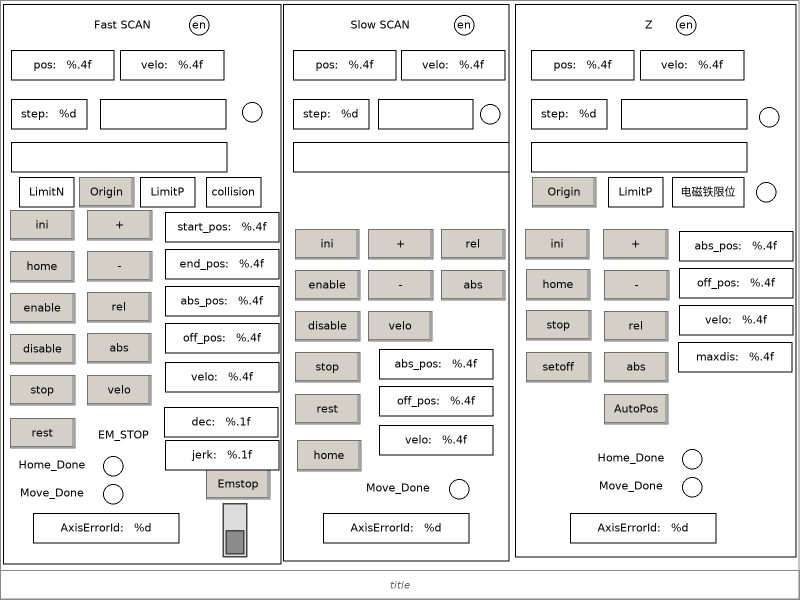
VISUALIZATION F1_AXIS  // 800x600
    RoundedRectangle (3,4 278x560)
    RoundedRectangle (515,4 281x553)
    RoundedRectangle (283,4 226x557)
    Button (87,210 65x30), "+", colour toggle: GVL_API.stAxis[1].JogForward
        tap GVL_API.stAxis[1].JogForward
    Button (87,251 65x30), "-", colour toggle: GVL_API.stAxis[1].JogBackwards
        tap GVL_API.stAxis[1].JogBackwards
    Button (10,251 64x31), "home", colour toggle: GVL_API.stAxis[1].homeExe
        toggle GVL_API.stAxis[1].homeExe
    Button (79,177 55x30), "Origin", colour toggle: Axis[1].IO.snHome
        toggle Axis[1].IO.snHome
    Rectangle (11,50 103x30), "pos: %.4f", text variable: Axis[1].Ref.NcToPlc.ActPos
    Rectangle (120,50 104x30), "velo: %.4f", text variable: Axis[1].Ref.NcToPlc.ActVelo
    Ellipse (189,15 20x20), "en", colour toggle: Axis[1].Ref.Status.ControlLoopClosed
    Button (87,292 64x30), "rel", colour toggle: GVL_API.stAxis[1].MoveRelativeExe
        toggle GVL_API.stAxis[1].MoveRelativeExe
    Button (87,333 64x30), "abs", colour toggle: GVL_API.stAxis[1].MoveAbsoluteExe
        toggle GVL_API.stAxis[1].MoveAbsoluteExe
    Button (87,375 64x30), "velo", colour toggle: GVL_API.stAxis[1].MoveConstantVelocity
        toggle GVL_API.stAxis[1].MoveConstantVelocity
    Button (10,210 64x30), "ini", colour toggle: GVL_API.stAxis[1].initialize
        toggle GVL_API.stAxis[1].initialize
    Button (10,375 65x30), "stop", colour toggle: GVL_API.stAxis[1].stop
        toggle GVL_API.stAxis[1].stop
    Rectangle (165,212 114x30), "start_pos: %.4f", text variable: GVL_API.stAxis[1].constantvelocitystart
        OnMouseDown: write GVL_API.stAxis[1].constantvelocitystart via Default
    Rectangle (165,249 114x30), "end_pos: %.4f", text variable: GVL_API.stAxis[1].constanvelocityend
        OnMouseDown: write GVL_API.stAxis[1].constanvelocityend via Default
    Rectangle (165,323 114x30), "off_pos: %.4f", text variable: GVL_API.stAxis[1].requestedoffset
        OnMouseDown: write GVL_API.stAxis[1].requestedoffset via Default
    Rectangle (165,286 114x30), "abs_pos: %.4f", text variable: GVL_API.stAxis[1].requestedposition
        OnMouseDown: write GVL_API.stAxis[1].requestedposition via Default
    Rectangle (165,362 114x30), "velo: %.4f", text variable: GVL_API.stAxis[1].velocity
        OnMouseDown: write GVL_API.stAxis[1].velocity via Default
    Rectangle (11,99 76x30), "step: %d", text variable: P_FastScan.SysStep
        OnMouseDown: write P_FastScan.SysStep via Default
    Button (10,418 65x30), "rest", colour toggle: GVL_API.stAxis[1].reset
        toggle GVL_API.stAxis[1].reset
    Button (10,293 65x30), "enable", colour toggle: GVL_API.stAxis[1].enabled
        toggle GVL_API.stAxis[1].enabled
    Rectangle (100,99 126x30), text list: 'TextList_xyzState', text index: GVL_API.stAxis[1].state
    Rectangle (11,142 216x30), text list: 'TextList_xyErrorid', text index: GVL_API.stAxis[1].ErrorId
    Button (206,469 64x30), "Emstop", colour toggle: GVL.Emstop_SAFE
    Label (70,10 105x30), "Fast SCAN"
    Button (368,229 65x30), "+", colour toggle: GVL_API.stAxis[2].JogForward
        tap GVL_API.stAxis[2].JogForward
    Button (368,270 65x30), "-", colour toggle: GVL_API.stAxis[2].JogBackwards
        tap GVL_API.stAxis[2].JogBackwards
    Rectangle (293,50 103x30), "pos: %.4f", text variable: Axis[2].Ref.NcToPlc.ActPos
    Rectangle (401,50 104x30), "velo: %.4f", text variable: Axis[2].Ref.NcToPlc.ActVelo
    Ellipse (454,15 20x20), "en", colour toggle: Axis[2].Ref.Status.ControlLoopClosed
    Button (441,229 64x30), "rel", colour toggle: GVL_API.stAxis[2].MoveRelativeExe
        toggle GVL_API.stAxis[2].MoveRelativeExe
    Button (441,270 64x30), "abs", colour toggle: GVL_API.stAxis[2].MoveAbsoluteExe
        toggle GVL_API.stAxis[2].MoveAbsoluteExe
    Button (368,311 64x30), "velo", colour toggle: GVL_API.stAxis[2].MoveConstantVelocity
        toggle GVL_API.stAxis[2].MoveConstantVelocity
    Button (295,229 64x30), "ini", colour toggle: GVL_API.stAxis[2].initialize
        toggle GVL_API.stAxis[2].initialize
    Button (295,352 65x30), "stop", colour toggle: GVL_API.stAxis[2].stop
        toggle GVL_API.stAxis[2].stop
    Rectangle (379,386 114x30), "off_pos: %.4f", text variable: GVL_API.stAxis[2].requestedoffset
        OnMouseDown: write GVL_API.stAxis[2].requestedoffset via Default
    Rectangle (379,349 114x30), "abs_pos: %.4f", text variable: GVL_API.stAxis[2].requestedposition
        OnMouseDown: write GVL_API.stAxis[2].requestedposition via Default
    Rectangle (379,425 114x30), "velo: %.4f", text variable: GVL_API.stAxis[2].velocity
        OnMouseDown: write GVL_API.stAxis[2].velocity via Default
    Rectangle (293,99 76x30), "step: %d", text variable: P_SlowScan.SysStep
        OnMouseDown: write P_SlowScan.SysStep via Default
    Button (295,394 65x30), "rest", colour toggle: GVL_API.stAxis[2].reset
        toggle GVL_API.stAxis[2].reset
    Rectangle (378,99 95x30), text list: 'TextList_xyzState', text index: GVL_API.stAxis[2].state
    Rectangle (293,142 216x30), text list: 'TextList_xyErrorid', text index: GVL_API.stAxis[2].ErrorId
    Label (326,10 108x30), "Slow SCAN"
    Button (603,229 65x30), "+", colour toggle: GVL_API.stAxis[3].JogForward
        tap GVL_API.stAxis[3].JogForward
    Button (604,270 65x30), "-", colour toggle: GVL_API.stAxis[3].JogBackwards
        tap GVL_API.stAxis[3].JogBackwards
    Button (526,269 64x31), "home", colour toggle: GVL_API.stAxis[3].homeExe
        toggle GVL_API.stAxis[3].homeExe
    Button (532,177 64x30), "Origin", colour toggle: Axis[3].IO.snHome
        toggle Axis[3].IO.snHome
    Rectangle (531,50 103x30), "pos: %.4f", text variable: Axis[3].Ref.NcToPlc.ActPos
    Rectangle (640,50 104x30), "velo: %.4f", text variable: Axis[3].Ref.NcToPlc.ActVelo
    Ellipse (676,15 20x20), "en", colour toggle: Axis[3].Ref.Status.ControlLoopClosed
    Button (604,311 64x30), "rel", colour toggle: GVL_API.stAxis[3].MoveRelativeExe
        toggle GVL_API.stAxis[3].MoveRelativeExe
    Button (604,352 64x30), "abs", colour toggle: GVL_API.stAxis[3].MoveAbsoluteExe
        toggle GVL_API.stAxis[3].MoveAbsoluteExe
    Button (604,394 64x30), "AutoPos", colour toggle: GVL_API.stAxis[1].MoveConstantVelocity
        toggle GVL_API.stAxis[3].Automatic_positioning
    Button (525,229 64x30), "ini", colour toggle: GVL_API.stAxis[3].initialize
        toggle GVL_API.stAxis[3].initialize
    Button (526,310 65x30), "stop", colour toggle: GVL_API.stAxis[3].stop
        toggle GVL_API.stAxis[3].stop
    Rectangle (679,268 114x30), "off_pos: %.4f", text variable: GVL_API.stAxis[3].requestedoffset
        OnMouseDown: write GVL_API.stAxis[3].requestedoffset via Default
    Rectangle (679,231 114x30), "abs_pos: %.4f", text variable: GVL_API.stAxis[3].requestedposition
        OnMouseDown: write GVL_API.stAxis[3].requestedposition via Default
    Rectangle (679,305 114x30), "velo: %.4f", text variable: GVL_API.stAxis[3].velocity
        OnMouseDown: write GVL_API.stAxis[3].velocity via Default
    Rectangle (531,99 76x30), "step: %d", text variable: P_Z_Axis.SysStep
        OnMouseDown: write P_Z_Axis.SysStep via Default
    Rectangle (621,99 126x30), text list: 'TextList_xyzState', text index: GVL_API.stAxis[3].state
    Rectangle (531,142 216x30), text list: 'TextList_zErrorid', text index: GVL_API.stAxis[3].ErrorId
    Label (609,10 80x30), "Z"
    Button (526,352 65x30), "setoff", colour toggle: GVL_API.stAxis[3].setoff
        toggle GVL_API.stAxis[3].setoff
    Rectangle (678,342 114x30), "maxdis: %.4f", text variable: GVL_API.stAxis[3].maxDistance
        OnMouseDown: write GVL_API.stAxis[3].maxDistance via Default
    Ellipse (756,182 20x20), colour toggle: stOutput.bqElectromagnet_power
    Rectangle (33,513 146x30), "AxisErrorId: %d", text variable: GVL_API.stAxis[1].AxisErrorId
    Rectangle (323,513 146x30), "AxisErrorId: %d", text variable: GVL_API.stAxis[2].AxisErrorId
    Rectangle (570,513 146x30), "AxisErrorId: %d", text variable: GVL_API.stAxis[2].AxisErrorId
    Button (10,334 65x30), "disable", colour toggle: GVL_API.stAxis[1].Disable
        toggle GVL_API.stAxis[1].Disable
    Button (295,270 65x30), "enable", colour toggle: GVL_API.stAxis[2].enabled
        toggle GVL_API.stAxis[2].enabled
    Button (295,311 65x30), "disable", colour toggle: GVL_API.stAxis[2].Disable
        toggle GVL_API.stAxis[2].Disable
    DipSwitch (208,503 54x54), variable: GVL.HMI_btEmstop, behaviour: TOGGLE, style: Switch-DipSwitch-Gray
    Frame (0,570 800x30)
        shows title()
    Rectangle (206,177 55x30), "collision", colour toggle: GVL.shuttle_crash
    Rectangle (140,177 55x30), "LimitP", colour toggle: Axis[1].IO.snLimitP
    Rectangle (19,177 55x30), "LimitN", colour toggle: Axis[1].IO.snLimitN
    Rectangle (608,177 55x30), "LimitP", colour toggle: Axis[3].IO.snLimitP
    Rectangle (672,177 72x30), "电磁铁限位", colour toggle: stInput.biElectromagnet_limit
    Ellipse (242,102 20x20), colour toggle: GVL_API.stAxis[1].Error
    Button (297,440 64x31), "home", colour toggle: GVL_API.stAxis[2].homeExe
        toggle GVL_API.stAxis[2].homeExe
    Ellipse (480,104 20x20), colour toggle: GVL_API.stAxis[2].Error
    Ellipse (759,107 20x20), colour toggle: GVL_API.stAxis[3].Error
    Ellipse (103,456 20x20), colour toggle: GVL_API.stAxis[1].Home_Done
    Label (12,450 80x30), "Home_Done"
    Label (12,478 80x30), "Move_Done"
    Ellipse (103,484 20x20), colour toggle: GVL_API.stAxis[1].Move_Done
    Label (358,473 80x30), "Move_Done"
    Ellipse (449,479 20x20), colour toggle: GVL_API.stAxis[2].Move_Done
    Label (591,471 80x30), "Move_Done"
    Ellipse (682,449 20x20), colour toggle: GVL_API.stAxis[3].Home_Done
    Label (591,443 80x30), "Home_Done"
    Ellipse (682,477 20x20), colour toggle: GVL_API.stAxis[3].Move_Done
    Rectangle (164,407 114x30), "dec: %.1f", text variable: HMI_EM_STOP_Dec_FS
        OnMouseDown: write HMI_EM_STOP_Dec_FS via Default
    Rectangle (165,440 114x30), "jerk: %.1f", text variable: HMI_EM_STOP_Jerk_FS
        OnMouseDown: write HMI_EM_STOP_Jerk_FS via Default
    Label (71,420 105x30), "EM_STOP"
END_VISUALIZATION

(* stored: Version 1.1.0.1, ProductVersion 3.1.4024.11
   Visu F1_AXIS: Id {ff8b43e9-deb7-4f5a-a8c5-5bcb609c40c8} *)
